// TIA Portal V20 export
FUNCTION "CallDiagnostic" : Void   // FC16, LAD
TITLE = Diagnose / Diagnostics
AUTHOR : SICAR
FAMILY : Diag
// Aufruf: Diagnose / Call of SICAR Diagnostic blocks
// stored: IsIECCheckEnabled true, SetENOAutomatically true
   VAR_TEMP
      statWStringName : WString[24];
      tempHardwareOKexample : Bool;   // REPLACE: This output can be used as an interlock for Control Modules
   END_VAR
   VAR CONSTANT
      TRUE : Bool := TRUE;
   END_VAR
   // Ret_Val : Ret_Val
   VAR_TEMP   // added for the SCL form of the ladder/FBD networks
      _w1 : Bool;
      _w2 : Bool;
   END_VAR
BEGIN

REGION Network 1: Beschreibung / BLOCK INFO HEADER
   // **Betriebsart Automatik / Hand**  
   // Der Baustein ist keiner Betriebsart / Betriebsartenbereich zugeordnet.  
   // 
   // **Alarme**  
   // Der Baustein generiert keine Alarme.  
   // 
   // #### PLC-Datentypen  
   // Verwendete PLC-Datentypen für den SPS-Programmbaustein und das zugehörige WinCC-Bild.  
   // 
   // {.pageWidth}
   // ![Image](CallInterfaceSignals/de/image1.PNG)
   //  
   //  
   // #### Bausteinaufrufe 
   // Der Baustein “LSicar_InterfaceSignalsBool“ wird in diesem FB als Multi-Instanz aufgerufen, entspr. nebenstehender beispielhafter Darstellung.  
   // 
   // {.pageWidth}
   // ![Image](CallInterfaceSignals/de/image2.PNG)
   //  
   // Um einen neuen FB aufzurufen, ziehen Sie den FB in ein neues Netzwerk, wählen Sie „Multiinstanz“ aus, vergeben Sie einen Namen und parametrieren Sie den FB-Aufruf.  
   // 
   // {.pageWidth}
   // ![Image](CallInterfaceSignals/de/image3.PNG)
   //  
   //  
   // #### Weitere Hinweise 
   // 
   // #### Updateinfo 
   // 
   // #### Weitere Dokumente 
   // 
   // ![Icon](_Icon/reference.PNG)
   // 
   // ..\Library Types\LSicar_InterfaceSignalsBool.pdf
   // SIEMENS AG / (c)Copyright 2023
   // ------------------------------------------------------------------------------
   // Title:            CallDiagnostic (FC16)
   // Comment/Function: Call of SICAR Diagnostic blocks
   // Library/Family:   Diag
   // Author:           SICAR
   // Tested with:      ---
   // Engineering:      TIA Portal V19
   // Restrictions:     -
   // Requirements:     ---
   // ------------------------------------------------------------------------------
   // Change log table:
   // Version | Date | Expert in charge | Changes applied
   // -------|---------|-------------|--------------------------------------------
   // 01.00.00 | 01.01.1999 | Person x | First released version
   // 01.00.01 | 02.01.1999 | Person y | Block was Updated
END_REGION

REGION Network 2: Call: Diagnostic Profinet Devices
   // For diagnose the whole profinet devices of this PLC
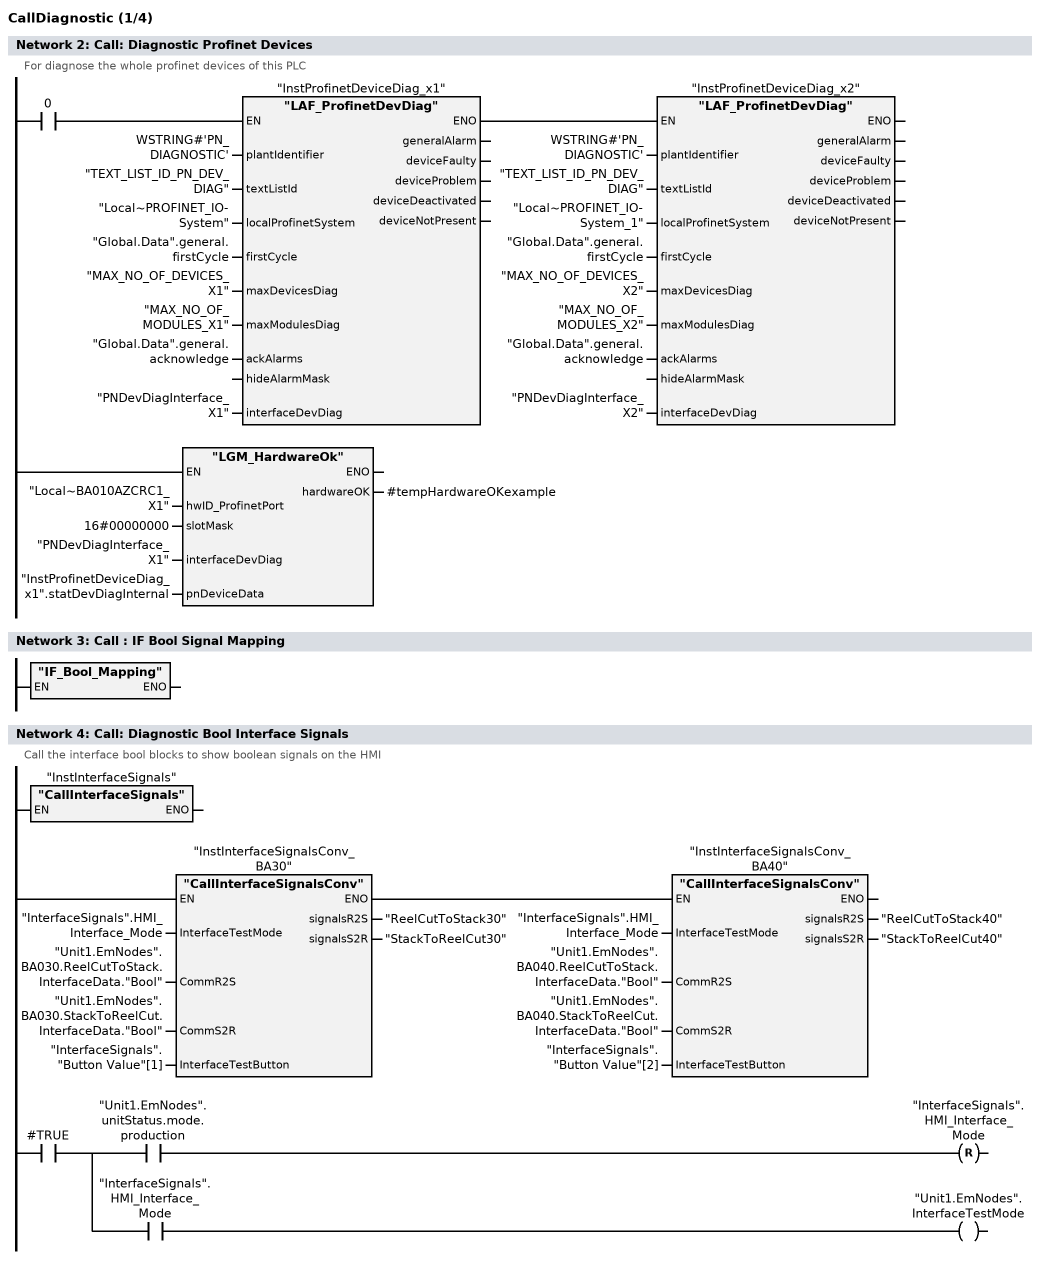
   RUNG wire#powerrail
      Contact( 0 )
      "InstProfinetDeviceDiag_x1"(plantIdentifier := WSTRING#'PN_DIAGNOSTIC', textListId := "TEXT_LIST_ID_PN_DEV_DIAG", localProfinetSystem := "Local~PROFINET_IO-System", firstCycle := "Global.Data".general.firstCycle, maxDevicesDiag := "MAX_NO_OF_DEVICES_X1", maxModulesDiag := "MAX_NO_OF_MODULES_X1", ackAlarms := "Global.Data".general.acknowledge, hideAlarmMask :=, interfaceDevDiag := "PNDevDiagInterface_X1", generalAlarm =>, deviceFaulty =>, deviceProblem =>, deviceDeactivated =>, deviceNotPresent =>)
      "InstProfinetDeviceDiag_x2"(plantIdentifier := WSTRING#'PN_DIAGNOSTIC', textListId := "TEXT_LIST_ID_PN_DEV_DIAG", localProfinetSystem := "Local~PROFINET_IO-System_1", firstCycle := "Global.Data".general.firstCycle, maxDevicesDiag := "MAX_NO_OF_DEVICES_X2", maxModulesDiag := "MAX_NO_OF_MODULES_X2", ackAlarms := "Global.Data".general.acknowledge, hideAlarmMask :=, interfaceDevDiag := "PNDevDiagInterface_X2", generalAlarm =>, deviceFaulty =>, deviceProblem =>, deviceDeactivated =>, deviceNotPresent =>)
   END_RUNG
   RUNG wire#powerrail
      "LGM_HardwareOk"(hwID_ProfinetPort := "Local~BA010AZCRC1_X1", slotMask := 16#00000000, interfaceDevDiag := "PNDevDiagInterface_X1", pnDeviceData := "InstProfinetDeviceDiag_x1".statDevDiagInternal, hardwareOK => #tempHardwareOKexample)
   END_RUNG
   // the same network as SCL:
   "InstProfinetDeviceDiag_x1"(EN := 0,   // "LAF_ProfinetDevDiag"
                           plantIdentifier := WSTRING#'PN_DIAGNOSTIC',
                           textListId := "TEXT_LIST_ID_PN_DEV_DIAG",
                           localProfinetSystem := "Local~PROFINET_IO-System",
                           firstCycle := "Global.Data".general.firstCycle,
                           maxDevicesDiag := "MAX_NO_OF_DEVICES_X1",
                           maxModulesDiag := "MAX_NO_OF_MODULES_X1",
                           ackAlarms := "Global.Data".general.acknowledge,
                           interfaceDevDiag := "PNDevDiagInterface_X1",
                           ENO => #_w1);
   IF #_w1 THEN
       "InstProfinetDeviceDiag_x2"(plantIdentifier := WSTRING#'PN_DIAGNOSTIC',   // "LAF_ProfinetDevDiag"
                               textListId := "TEXT_LIST_ID_PN_DEV_DIAG",
                               localProfinetSystem := "Local~PROFINET_IO-System_1",
                               firstCycle := "Global.Data".general.firstCycle,
                               maxDevicesDiag := "MAX_NO_OF_DEVICES_X2",
                               maxModulesDiag := "MAX_NO_OF_MODULES_X2",
                               ackAlarms := "Global.Data".general.acknowledge,
                               interfaceDevDiag := "PNDevDiagInterface_X2");
   END_IF;
   "LGM_HardwareOk"(hwID_ProfinetPort := "Local~BA010AZCRC1_X1",
                    slotMask := 16#00000000,
                    interfaceDevDiag := "PNDevDiagInterface_X1",
                    pnDeviceData := "InstProfinetDeviceDiag_x1".statDevDiagInternal,
                    hardwareOK => #tempHardwareOKexample);
END_REGION

REGION Network 3: Call : IF Bool Signal Mapping
   RUNG wire#powerrail
      "IF_Bool_Mapping"()
   END_RUNG
   // the same network as SCL:
   "IF_Bool_Mapping"();
END_REGION

REGION Network 4: Call: Diagnostic Bool Interface Signals
   // Call the interface bool blocks to show boolean signals on the HMI
   RUNG wire#powerrail
      "InstInterfaceSignals"()
   END_RUNG
   RUNG wire#powerrail
      "InstInterfaceSignalsConv_BA30"(InterfaceTestMode := "InterfaceSignals".HMI_Interface_Mode, CommR2S := "Unit1.EmNodes".BA030.ReelCutToStack.InterfaceData."Bool", CommS2R := "Unit1.EmNodes".BA030.StackToReelCut.InterfaceData."Bool", InterfaceTestButton := "InterfaceSignals"."Button Value"[1], signalsR2S => "ReelCutToStack30", signalsS2R => "StackToReelCut30")
      "InstInterfaceSignalsConv_BA40"(InterfaceTestMode := "InterfaceSignals".HMI_Interface_Mode, CommR2S := "Unit1.EmNodes".BA040.ReelCutToStack.InterfaceData."Bool", CommS2R := "Unit1.EmNodes".BA040.StackToReelCut.InterfaceData."Bool", InterfaceTestButton := "InterfaceSignals"."Button Value"[2], signalsR2S => "ReelCutToStack40", signalsS2R => "StackToReelCut40")
   END_RUNG
   RUNG wire#powerrail
      Contact( #TRUE )
      wire#w1
      Contact( "Unit1.EmNodes".unitStatus.mode.production )
      R_Coil( "InterfaceSignals".HMI_Interface_Mode )
   END_RUNG
   RUNG wire#w1
      Contact( "InterfaceSignals".HMI_Interface_Mode )
      Coil( "Unit1.EmNodes".InterfaceTestMode )
   END_RUNG
   // the same network as SCL:
   "InstInterfaceSignals"();   // "CallInterfaceSignals"
   "InstInterfaceSignalsConv_BA30"(InterfaceTestMode := "InterfaceSignals".HMI_Interface_Mode,   // "CallInterfaceSignalsConv"
                           CommR2S := "Unit1.EmNodes".BA030.ReelCutToStack.InterfaceData."Bool",
                           CommS2R := "Unit1.EmNodes".BA030.StackToReelCut.InterfaceData."Bool",
                           InterfaceTestButton := "InterfaceSignals"."Button Value"[1],
                           signalsR2S => "ReelCutToStack30",
                           signalsS2R => "StackToReelCut30",
                           ENO => #_w1);
   IF #_w1 THEN
       "InstInterfaceSignalsConv_BA40"(InterfaceTestMode := "InterfaceSignals".HMI_Interface_Mode,   // "CallInterfaceSignalsConv"
                               CommR2S := "Unit1.EmNodes".BA040.ReelCutToStack.InterfaceData."Bool",
                               CommS2R := "Unit1.EmNodes".BA040.StackToReelCut.InterfaceData."Bool",
                               InterfaceTestButton := "InterfaceSignals"."Button Value"[2],
                               signalsR2S => "ReelCutToStack40",
                               signalsS2R => "StackToReelCut40");
   END_IF;
   IF #TRUE AND "Unit1.EmNodes".unitStatus.mode.production THEN
       "InterfaceSignals".HMI_Interface_Mode := FALSE;
   END_IF;
   "Unit1.EmNodes".InterfaceTestMode := #TRUE AND "InterfaceSignals".HMI_Interface_Mode;
END_REGION

REGION Network 5: Call: Diagnostics Drives
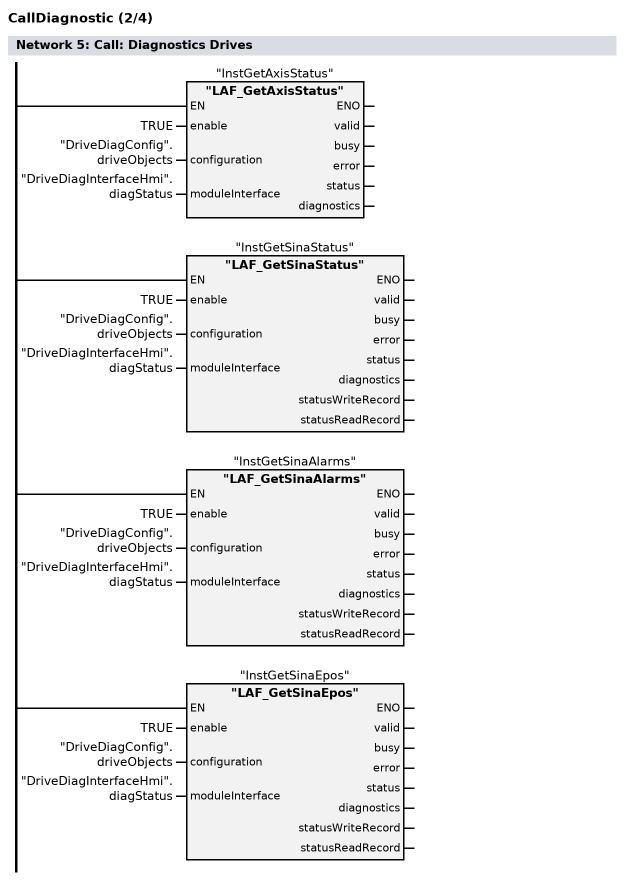
   RUNG wire#powerrail
      "InstGetAxisStatus"(enable := TRUE, configuration := "DriveDiagConfig".driveObjects, moduleInterface := "DriveDiagInterfaceHmi".diagStatus, valid =>, busy =>, error =>, status =>, diagnostics =>)
   END_RUNG
   RUNG wire#powerrail
      "InstGetSinaStatus"(enable := TRUE, configuration := "DriveDiagConfig".driveObjects, moduleInterface := "DriveDiagInterfaceHmi".diagStatus, valid =>, busy =>, error =>, status =>, diagnostics =>, statusWriteRecord =>, statusReadRecord =>)
   END_RUNG
   RUNG wire#powerrail
      "InstGetSinaAlarms"(enable := TRUE, configuration := "DriveDiagConfig".driveObjects, moduleInterface := "DriveDiagInterfaceHmi".diagStatus, valid =>, busy =>, error =>, status =>, diagnostics =>, statusWriteRecord =>, statusReadRecord =>)
   END_RUNG
   RUNG wire#powerrail
      "InstGetSinaEpos"(enable := TRUE, configuration := "DriveDiagConfig".driveObjects, moduleInterface := "DriveDiagInterfaceHmi".diagStatus, valid =>, busy =>, error =>, status =>, diagnostics =>, statusWriteRecord =>, statusReadRecord =>)
   END_RUNG
   // the same network as SCL:
   "InstGetAxisStatus"(enable := TRUE,   // "LAF_GetAxisStatus"
                       configuration := "DriveDiagConfig".driveObjects,
                       moduleInterface := "DriveDiagInterfaceHmi".diagStatus);
   "InstGetSinaStatus"(enable := TRUE,   // "LAF_GetSinaStatus"
                       configuration := "DriveDiagConfig".driveObjects,
                       moduleInterface := "DriveDiagInterfaceHmi".diagStatus);
   "InstGetSinaAlarms"(enable := TRUE,   // "LAF_GetSinaAlarms"
                       configuration := "DriveDiagConfig".driveObjects,
                       moduleInterface := "DriveDiagInterfaceHmi".diagStatus);
   "InstGetSinaEpos"(enable := TRUE,   // "LAF_GetSinaEpos"
                     configuration := "DriveDiagConfig".driveObjects,
                     moduleInterface := "DriveDiagInterfaceHmi".diagStatus);
END_REGION

REGION Network 6: Call: Diagnostics Ident RFID
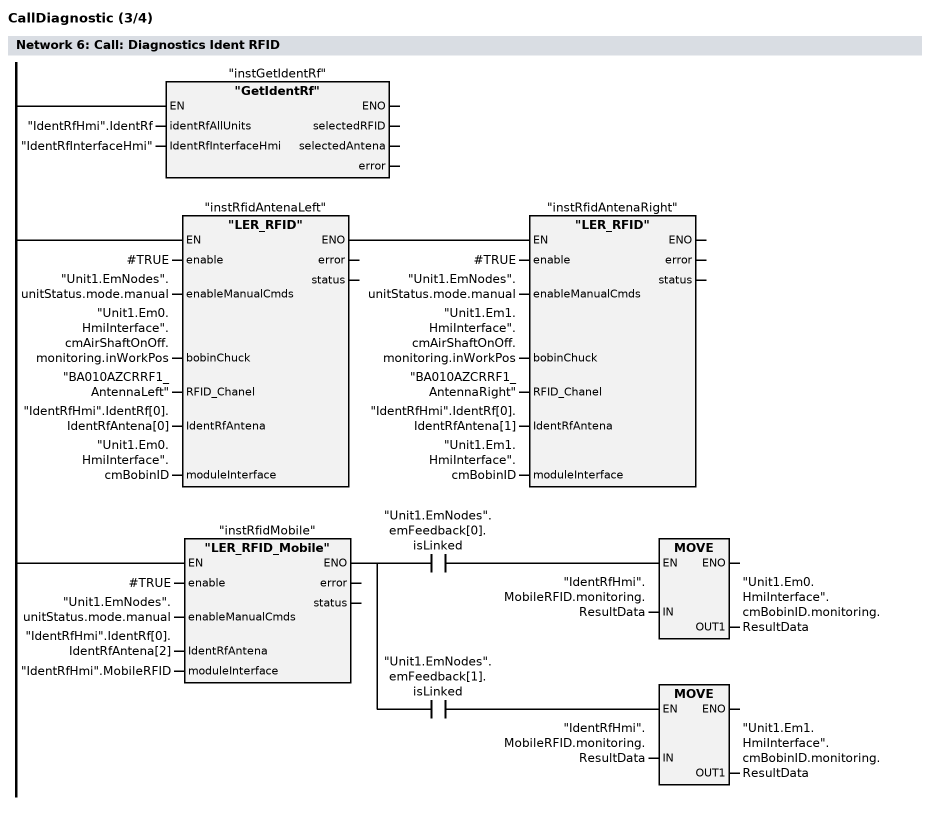
   RUNG wire#powerrail
      "instGetIdentRf"(identRfAllUnits := "IdentRfHmi".IdentRf, IdentRfInterfaceHmi := "IdentRfInterfaceHmi", selectedRFID =>, selectedAntena =>, error =>)
   END_RUNG
   RUNG wire#powerrail
      "instRfidAntenaLeft"(enable := #TRUE, enableManualCmds := "Unit1.EmNodes".unitStatus.mode.manual, bobinChuck := "Unit1.Em0.HmiInterface".cmAirShaftOnOff.monitoring.inWorkPos, RFID_Chanel := "BA010AZCRRF1_AntennaLeft", IdentRfAntena := "IdentRfHmi".IdentRf[0].IdentRfAntena[0], moduleInterface := "Unit1.Em0.HmiInterface".cmBobinID, error =>, status =>)
      "instRfidAntenaRight"(enable := #TRUE, enableManualCmds := "Unit1.EmNodes".unitStatus.mode.manual, bobinChuck := "Unit1.Em1.HmiInterface".cmAirShaftOnOff.monitoring.inWorkPos, RFID_Chanel := "BA010AZCRRF1_AntennaRight", IdentRfAntena := "IdentRfHmi".IdentRf[0].IdentRfAntena[1], moduleInterface := "Unit1.Em1.HmiInterface".cmBobinID, error =>, status =>)
   END_RUNG
   RUNG wire#powerrail
      "instRfidMobile"(enable := #TRUE, enableManualCmds := "Unit1.EmNodes".unitStatus.mode.manual, IdentRfAntena := "IdentRfHmi".IdentRf[0].IdentRfAntena[2], moduleInterface := "IdentRfHmi".MobileRFID, error =>, status =>)
      wire#w1
      Contact( "Unit1.EmNodes".emFeedback[0].isLinked )
      Move(in := "IdentRfHmi".MobileRFID.monitoring.ResultData, out1 => "Unit1.Em0.HmiInterface".cmBobinID.monitoring.ResultData)
   END_RUNG
   RUNG wire#w1
      Contact( "Unit1.EmNodes".emFeedback[1].isLinked )
      Move(in := "IdentRfHmi".MobileRFID.monitoring.ResultData, out1 => "Unit1.Em1.HmiInterface".cmBobinID.monitoring.ResultData)
   END_RUNG
   // the same network as SCL:
   "instGetIdentRf"(identRfAllUnits := "IdentRfHmi".IdentRf, IdentRfInterfaceHmi := "IdentRfInterfaceHmi");   // "GetIdentRf"
   "instRfidAntenaLeft"(enable := #TRUE,   // "LER_RFID"
                        enableManualCmds := "Unit1.EmNodes".unitStatus.mode.manual,
                        bobinChuck := "Unit1.Em0.HmiInterface".cmAirShaftOnOff.monitoring.inWorkPos,
                        RFID_Chanel := "BA010AZCRRF1_AntennaLeft",
                        IdentRfAntena := "IdentRfHmi".IdentRf[0].IdentRfAntena[0],
                        moduleInterface := "Unit1.Em0.HmiInterface".cmBobinID,
                        ENO => #_w1);
   IF #_w1 THEN
       "instRfidAntenaRight"(enable := #TRUE,   // "LER_RFID"
                             enableManualCmds := "Unit1.EmNodes".unitStatus.mode.manual,
                             bobinChuck := "Unit1.Em1.HmiInterface".cmAirShaftOnOff.monitoring.inWorkPos,
                             RFID_Chanel := "BA010AZCRRF1_AntennaRight",
                             IdentRfAntena := "IdentRfHmi".IdentRf[0].IdentRfAntena[1],
                             moduleInterface := "Unit1.Em1.HmiInterface".cmBobinID);
   END_IF;
   "instRfidMobile"(enable := #TRUE,   // "LER_RFID_Mobile"
                    enableManualCmds := "Unit1.EmNodes".unitStatus.mode.manual,
                    IdentRfAntena := "IdentRfHmi".IdentRf[0].IdentRfAntena[2],
                    moduleInterface := "IdentRfHmi".MobileRFID,
                    ENO => #_w2);
   IF #_w2 AND "Unit1.EmNodes".emFeedback[0].isLinked THEN
       "Unit1.Em0.HmiInterface".cmBobinID.monitoring.ResultData := "IdentRfHmi".MobileRFID.monitoring.ResultData;
   END_IF;
   IF #_w2 AND "Unit1.EmNodes".emFeedback[1].isLinked THEN
       "Unit1.Em1.HmiInterface".cmBobinID.monitoring.ResultData := "IdentRfHmi".MobileRFID.monitoring.ResultData;
   END_IF;
END_REGION

REGION Network 7: Call: TraceCode Generation
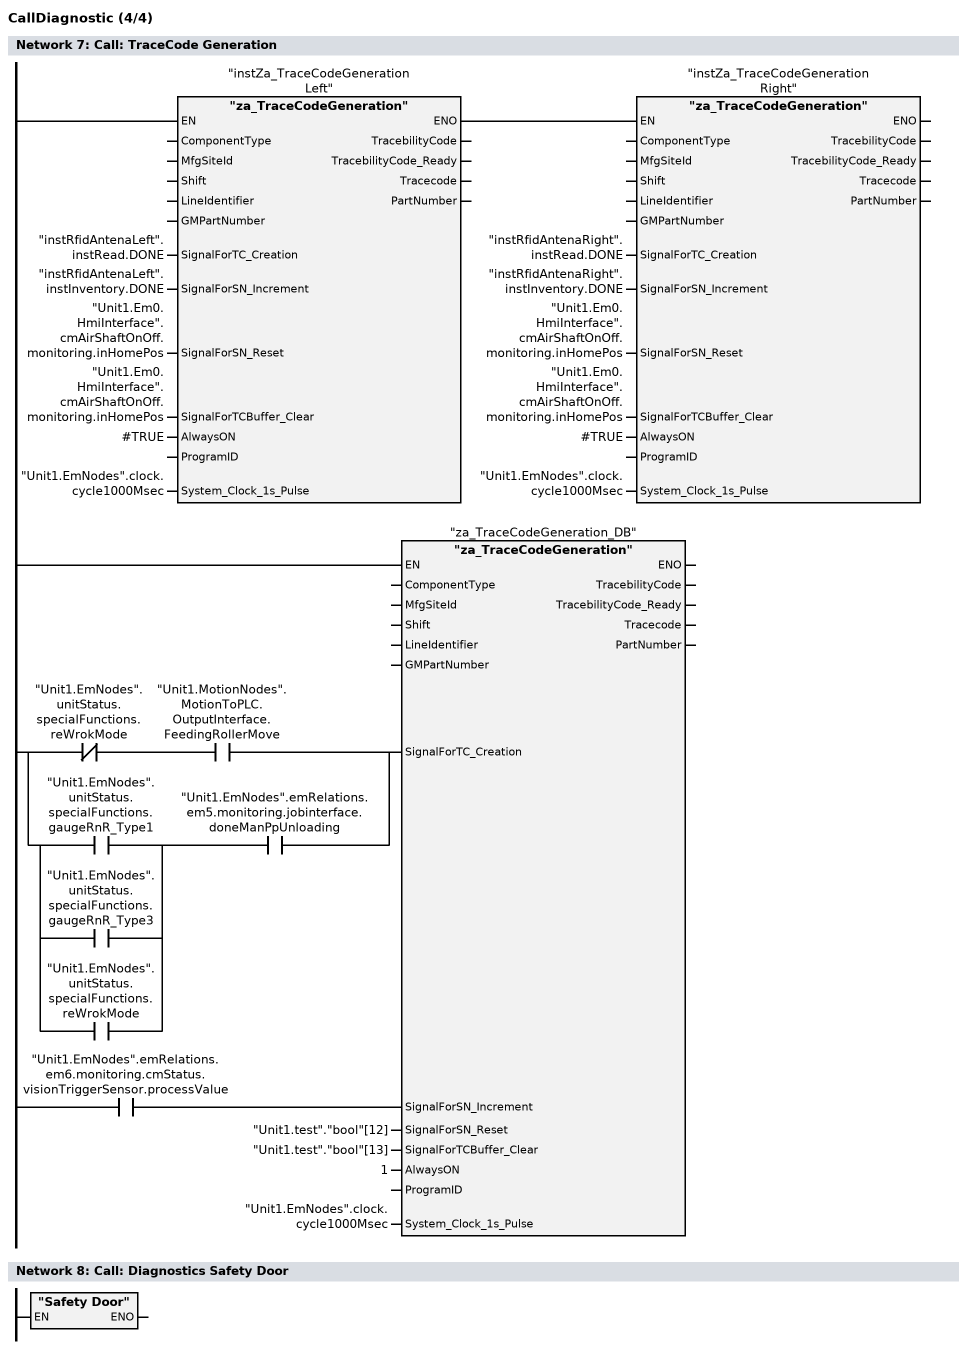
   RUNG wire#powerrail
      "instZa_TraceCodeGenerationLeft"(ComponentType :=, MfgSiteId :=, Shift :=, LineIdentifier :=, GMPartNumber :=, SignalForTC_Creation := "instRfidAntenaLeft".instRead.DONE, SignalForSN_Increment := "instRfidAntenaLeft".instInventory.DONE, SignalForSN_Reset := "Unit1.Em0.HmiInterface".cmAirShaftOnOff.monitoring.inHomePos, SignalForTCBuffer_Clear := "Unit1.Em0.HmiInterface".cmAirShaftOnOff.monitoring.inHomePos, AlwaysON := #TRUE, ProgramID :=, System_Clock_1s_Pulse := "Unit1.EmNodes".clock.cycle1000Msec, TracebilityCode =>, TracebilityCode_Ready =>, Tracecode =>, PartNumber =>)
      "instZa_TraceCodeGenerationRight"(ComponentType :=, MfgSiteId :=, Shift :=, LineIdentifier :=, GMPartNumber :=, SignalForTC_Creation := "instRfidAntenaRight".instRead.DONE, SignalForSN_Increment := "instRfidAntenaRight".instInventory.DONE, SignalForSN_Reset := "Unit1.Em0.HmiInterface".cmAirShaftOnOff.monitoring.inHomePos, SignalForTCBuffer_Clear := "Unit1.Em0.HmiInterface".cmAirShaftOnOff.monitoring.inHomePos, AlwaysON := #TRUE, ProgramID :=, System_Clock_1s_Pulse := "Unit1.EmNodes".clock.cycle1000Msec, TracebilityCode =>, TracebilityCode_Ready =>, Tracecode =>, PartNumber =>)
   END_RUNG
   RUNG wire#powerrail
      "za_TraceCodeGeneration_DB"(SignalForTC_Creation := wire#w2, SignalForSN_Increment := wire#w3, ComponentType :=, MfgSiteId :=, Shift :=, LineIdentifier :=, GMPartNumber :=, SignalForSN_Reset := "Unit1.test"."bool"[12], SignalForTCBuffer_Clear := "Unit1.test"."bool"[13], AlwaysON := 1, ProgramID :=, System_Clock_1s_Pulse := "Unit1.EmNodes".clock.cycle1000Msec, TracebilityCode =>, TracebilityCode_Ready =>, Tracecode =>, PartNumber =>)
   END_RUNG
   RUNG wire#powerrail
      I_Contact( "Unit1.EmNodes".unitStatus.specialFunctions.reWrokMode )
      Contact( "Unit1.MotionNodes".MotionToPLC.OutputInterface.FeedingRollerMove )
   END_RUNG wire#w2
   RUNG wire#powerrail
      Contact( "Unit1.EmNodes".unitStatus.specialFunctions.gaugeRnR_Type1 )
      wire#w1
      Contact( "Unit1.EmNodes".emRelations.em5.monitoring.jobinterface.doneManPpUnloading )
   END_RUNG wire#w2
   RUNG wire#powerrail
      Contact( "Unit1.EmNodes".unitStatus.specialFunctions.gaugeRnR_Type3 )
   END_RUNG wire#w1
   RUNG wire#powerrail
      Contact( "Unit1.EmNodes".unitStatus.specialFunctions.reWrokMode )
   END_RUNG wire#w1
   RUNG wire#powerrail
      Contact( "Unit1.EmNodes".emRelations.em6.monitoring.cmStatus.visionTriggerSensor.processValue )
   END_RUNG wire#w3
   // the same network as SCL:
   "instZa_TraceCodeGenerationLeft"(SignalForTC_Creation := "instRfidAntenaLeft".instRead.DONE,   // "za_TraceCodeGeneration"
                           SignalForSN_Increment := "instRfidAntenaLeft".instInventory.DONE,
                           SignalForSN_Reset := "Unit1.Em0.HmiInterface".cmAirShaftOnOff.monitoring.inHomePos,
                           SignalForTCBuffer_Clear := "Unit1.Em0.HmiInterface".cmAirShaftOnOff.monitoring.inHomePos,
                           AlwaysON := #TRUE,
                           System_Clock_1s_Pulse := "Unit1.EmNodes".clock.cycle1000Msec,
                           ENO => #_w1);
   IF #_w1 THEN
       "instZa_TraceCodeGenerationRight"(SignalForTC_Creation := "instRfidAntenaRight".instRead.DONE,   // "za_TraceCodeGeneration"
                               SignalForSN_Increment := "instRfidAntenaRight".instInventory.DONE,
                               SignalForSN_Reset := "Unit1.Em0.HmiInterface".cmAirShaftOnOff.monitoring.inHomePos,
                               SignalForTCBuffer_Clear := "Unit1.Em0.HmiInterface".cmAirShaftOnOff.monitoring.inHomePos,
                               AlwaysON := #TRUE,
                               System_Clock_1s_Pulse := "Unit1.EmNodes".clock.cycle1000Msec);
   END_IF;
   "za_TraceCodeGeneration_DB"(SignalForTC_Creation := (NOT "Unit1.EmNodes".unitStatus.specialFunctions.reWrokMode AND "Unit1.MotionNodes".MotionToPLC.OutputInterface.FeedingRollerMove) OR (("Unit1.EmNodes".unitStatus.specialFunctions.gaugeRnR_Type1 OR "Unit1.EmNodes".unitStatus.specialFunctions.gaugeRnR_Type3 OR "Unit1.EmNodes".unitStatus.specialFunctions.reWrokMode) AND "Unit1.EmNodes".emRelations.em5.monitoring.jobinterface.doneManPpUnloading),   // "za_TraceCodeGeneration"
                           SignalForSN_Increment := "Unit1.EmNodes".emRelations.em6.monitoring.cmStatus.visionTriggerSensor.processValue,
                           SignalForSN_Reset := "Unit1.test"."bool"[12],
                           SignalForTCBuffer_Clear := "Unit1.test"."bool"[13],
                           AlwaysON := 1,
                           System_Clock_1s_Pulse := "Unit1.EmNodes".clock.cycle1000Msec);
END_REGION

REGION Network 8: Call: Diagnostics Safety Door
   RUNG wire#powerrail
      "Safety Door"()
   END_RUNG
   // the same network as SCL:
   "Safety Door"();
END_REGION
END_FUNCTION
